// TIA Portal V16 export
// export: Created 2024-05-13T12:47:23.3777086Z, ExportSetting WithDefaults, DisplayName Totally Integrated Automation Portal, DisplayVersion V16 Update 6, DisplayName TIA Portal Version Control Interface, DisplayVersion V16 Update 2, DisplayName TIA Portal Openness, DisplayVersion V16 Update 6, DisplayName TIA Portal Test Suite Advanced, DisplayVersion V16, DisplayName SINAMICS Startdrive Advanced, DisplayVersion V16 Update 5, DisplayName SINAMICS Startdrive G130, G150, S120, S150, SINAMICS MV, S210, DisplayVersion V16 Update 5, DisplayName SINAMICS Startdrive G110M, G120, G120C, G120D, G120P, G115D, DisplayVersion V16 Update 5, DisplayName STEP 7 Professional, DisplayVersion V16 Update 6, DisplayName STEP 7 Safety, DisplayVersion V16, DisplayName WinCC Advanced, DisplayVersion V16 Update 6
TYPE "SCA_inkjetMarker_IO_Input"
// stored: IsFailsafeCompliant false
   STRUCT
      Safety_switch : Bool;   // Safety switch
      Arm_up : Bool;   // Arm up
      Arm_down : Bool;   // Arm down
      Pulse_A : Bool;   // Pulse A
      Pulse_B : Bool;   // Pulse B
      Area_free_1 : Bool;   // Area free 1
      Area_free_2 : Bool;   // Area free 2
      Man_arm_up : Bool;   // Manual up switch
      Man_arm_down : Bool;   // Manual down switch
      Close_to_roll : Bool;   // Print head close to roll
      Roll_sensing_1 : Bool;   // Roll sensing 1
      Roll_sensing_2 : Bool;   // Roll sensing 2
   END_STRUCT;
END_TYPE
